{attribute 'qualified_only'}
{attribute 'strict'}
TYPE E_CAMERA_State :
(
	IDLE,
	CONNECT,
	SEND,
	RECEIVE,
	DISCONNECT,
	//CHECKOS,
	BROWSEDIAG,
	BROWSELIVE,
	IMAGE,
	DECODE,
	HEARTBEAT,
	DONE
);
END_TYPE

(* stored: Version 1.1.0.1
   DUT E_CAMERA_State: Id {978fbf49-8c2c-4fcd-bf42-7e077b43f7d7} *)
